TYPE ref_cav :
STRUCT
	cav : ARRAY [1..8] OF  ref_palletize;
END_STRUCT
END_TYPE

(* stored: Version 1.1.0.1, ProductVersion 3.1.4024.11
   DUT ref_cav: Id {ff3324c6-b544-41fa-b72e-0b8e7252dd61} *)
